{attribute 'GeneratedUsingTerminal: AT2050-0501-0019'}
{attribute addProperty BoxType "AT2050-0501-0019"}
{attribute addProperty Id "A_0081_AT2002_5250_0018_AT2002_5250AT2002_33A3DF1B80"}
{attribute addProperty CRC "270884774"}
{attribute addProperty Size "80"}
TYPE A_0069_AT2050_0501_0019_AT2050_0501_10255FA6 EXTENDS AT2050_2EA6C9BF :
STRUCT
	{attribute addProperty Name "A_0081(AT2002-5250-0018) (AT2002-5250)"}
	{attribute addProperty PreviousPort "A_0069(AT2050-0501-0019) (AT2050-0501) : B"}
	A_0081_AT2002_5250_0018_AT2002_5250 : AT2002_33A3DF1B;
END_STRUCT
END_TYPE

(* stored: Version 1.2.0.0, ProductVersion 3.1.4024.9
   DUT A_0069_AT2050_0501_0019_AT2050_0501_10255FA6: Id {f846fbc5-16d2-4d44-b578-6d36cd4a94cc} *)
